// TIA Portal V17 export
// export: Created 2025-03-07T09:19:54.7926162Z, ExportSetting WithDefaults, DisplayName Totally Integrated Automation Portal, DisplayVersion V17 Update 8, DisplayName TIA Portal Openness, DisplayVersion V17 Update 8, DisplayName TIA Portal Version Control Interface, DisplayVersion V17, DisplayName SINAMICS Startdrive Advanced, DisplayVersion V17 SP2, DisplayName SINAMICS Startdrive G110M, G120, G120C, G120D, G120P, G115D, DisplayVersion V17 SP2, DisplayName SINAMICS Startdrive G130, G150, S120, S150, SINAMICS MV, S210, DisplayVersion V17 SP2, DisplayName STEP 7 Professional, DisplayVersion V17 Update 8, DisplayName SINUMERIK ONE STEP 7 Toolbox, DisplayVersion V17 Update 12, DisplayName SINUMERIK 840D sl STEP 7 Toolbox, DisplayVersion V17 Update 12, DisplayName STEP 7 Safety, DisplayVersion V17 Update 6, DisplayName WinCC Advanced, DisplayVersion V17 Update 8
TYPE "ABB_OUTPUTS"
// stored: IsFailsafeCompliant false
   STRUCT
      SYSTEM_SIGNAL : Struct
         SYS_MOTOR_ON : Bool;   // MACHINE HEARTBEAT (MACHINE TO GANTRY) / MOTORS ON STATE
         SYS_MOTOR_OFF : Bool;   // MOTORS OFF STATE
         SYS_CYCLE_ON : Bool;   // MACHINE EMERGENCY STOP OK (MACHINE TO GANTRY) / ROBOT IN CYCLE ON STATE
         SYS_AUTO_ON : Bool;   // MACHINE SAFETY GATES OK (LOCKED)(MACHINE TO GANTRY) / ROBOT IN AUTO MODE
         SYS_EMERG_UOP : Bool;   // MACHINE IN MANUAL MODE (MACHINE TO GANTRY) / EMERGENCY STOP ACTIVE
         SYS_ERROR : Bool;   // MACHINE IN AUTO MODE(MACHINE TO GANTRY) / EXECUTION ERROR ACTIVE
         SPARE_0_6 : Bool;   // MACHINE AUTO CYCLE RUNNING (MACHINE TO GANTRY)
         SPARE_0_7 : Bool;   // MACHINE IS IN WARMUP CYCLE (MACHINE TO GANTRY)
         SPARE_1_0 : Byte;   // MACHINE IN RUN OUT MODE (MACHINE TO GANTRY)
         SPARE_2_0 : Byte;   // MACHINE PART DEMAND SOON (MACHINE TO GANTRY)
         SPARE_3_0 : Byte;
      END_STRUCT;
      GENERAL_SIGNAL : Struct
         STYLE_INIT_ACK : Bool;   // GANTRY HEARTBEAT (GANTRY TO MACHINE) / ACKNOWLEDGE INITIATE STYLE
         IN_CYCLE : Bool;   // IN CYCLE
         REQ_TO_CONT : Bool;   // GANTRY EMERGENCY STOP OK (GANTRY TO MACHINE) / REQUEST TO CONTINUE
         DRY_CYCLE : Bool;   // DRY CYCLE MODE
         RBT_100_SPD : Bool;   // GANTRY IN MANUAL MODE (GANTRY TO MACHINE) / ROBOT 100% SPEED
         RBT_HEARTBEAT : Bool;   // GANTRY IN AUTO MODE (GANTRY TO MACHINE) / ROBOT HEARTBEAT SIGNAL
         "OP_PANEL_E-STOP" : Bool;   // GANTRY IN AUTO CYCLE RUNNING (GANTRY TO MACHINE) / OPERATOR PANEL E-STOP
         "TEACH_PENDANT_E-STOP" : Bool;   // GANTRY OVERHEAD DOOR CLOSED & LOCKED (GANTRY TO MACHINE) / TEACH PENDANT E-STOP
         EXT_ENABLED : Bool;   // GANTRY IN RUN OUT COMPLETE(GANTRY TO MACHINE) / EXTERNAL E-STOP
         DEAD_ENABLED : Bool;   // GANTRY CLEAR OF MACHINE (GANTRY TO MACHINE) / DEADMAN E-STOP
         "I/O_SIMULATE" : Bool;   // GANTRY CLEAR OF FIXTURE (GANTRY TO MACHINE) / I/O SIMULATED
         SRV_DISC_OFF : Bool;   // SERVO DISABLED OFF
         SRV_BATT_ALARM : Bool;   // LOW BATTERY ALARM ON SERVO
         TASK_OK : Bool;   // TASK OK
         STEP_MODE_ON : Bool;   // STEP MODE STATUS
         AUTO_MODE_ON : Bool;   // SELECTOR SWITCH IS SET TO AUTO
         MANUAL_ON : Bool;   // SELECTOR SWITCH IS SET TO MANUAL
         FENCE_OPEN : Bool;   // FENCE IS OPEN
         INTERLOCK : Bool;   // ROBOT IN INTERLOCK
         ROUT_ACTIVE : Bool;   // ROUTER ACTIVE BIT
         FAULT_RSP_ACK : Bool;   // HMI OPTION FAULT RESPONSE
         DCS_SIGN_MATCH : Bool;   // DCS SIGNATURE MATCH
         REQ_DEC_CODE : Bool;   // REQUEST DECITION
         FLT_TASK_UOPPED : Bool;   // ROBOT TASK STOPPED
         FLT_COLLISION : Bool;   // ROBOT COLLITION FAULT
         FLT_BAD_PLC_INPUT : Bool;   // BAD PLC INPUT
         FLT_GRIP_LOW_PRS : Bool;   // ROBOT GRIPPER PRESSURE LOW
         FLT_BAD_OPTN : Bool;   // BAD PLC FAULT RESPONSE
         RECOV_AT_MAIN : Bool;   // RECOVERY POINTER TO MAIN
         FLT_USER_BIT_8 : Bool;   // USER DEFINABLE FAULT BIT
         SPARE_7_6 : Bool;
         SPARE_7_7 : Bool;
         SPARE_8_0 : Byte;
         SPARE_9_0 : Byte;
      END_STRUCT;
      PROGRAM : Struct
         STYLE_PROGRAM_ACK : Byte;   // GANTRY HEARTBEAT (GANTRY TO MACHINE) / SELECT STYLE PROGRAM ACKNOWLEDGE
         DEC_CODE_ACK : Byte;   // SELECT DECITION CODE ACKNOWLEDGE
         PART_TYPE_ACK : Byte;   // GANTRY EMERGENCY STOP OK (GANTRY TO MACHINE) / PART TYPE ACKNOWLEDGE
         SPARE_13_0 : Byte;   // GANTRY EMERGENCY STOP OK (GANTRY TO MACHINE)
      END_STRUCT;
      GRIPPERS : Struct
         T1_GRIPPER_A_OPEN_REQ : Bool;   // ROBOT TOOL 1 GRIPPER A OPEN REQUEST
         T1_GRIPPER_A_CLOSE_REQ : Bool;   // ROBOT TOOL 1 GRIPPER A CLOSE REQUEST
         SPARE_14_2 : Bool;
         SPARE_14_3 : Bool;
         T1_GRIPPER_A_OPEN : Bool;   // ROBOT TOOL 1 GRIPPER A OPEN
         T1_GRIPPER_A_CLOSED : Bool;   // ROBOT TOOL 1 GRIPPER A CLOSED
         SPARE_14_6 : Bool;
         SPARE_14_7 : Bool;
         T1_GRIPPER_B_OPEN_REQ : Bool;   // ROBOT TOOL 1 GRIPPER B OPEN REQUEST
         T1_GRIPPER_B_CLOSE_REQ : Bool;   // ROBOT TOOL 1 GRIPPER B CLOSE REQUEST
         SPARE_15_2 : Bool;
         SPARE_15_3 : Bool;
         T1_GRIPPER_B_OPEN : Bool;   // ROBOT TOOL 1 GRIPPER B OPEN
         T1_GRIPPER_B_CLOSED : Bool;   // ROBOT TOOL 1 GRIPPER B CLOSED
         SPARE_15_6 : Bool;
         SPARE_15_7 : Bool;
         T1_GRIPPER_C_OPEN_REQ : Bool;   // ROBOT TOOL 1 GRIPPER C OPEN REQUEST
         T1_GRIPPER_C_CLOSE_REQ : Bool;   // ROBOT TOOL 1 GRIPPER C CLOSE REQUEST
         SPARE_16_2 : Bool;
         SPARE_16_3 : Bool;
         T1_GRIPPER_C_OPEN : Bool;   // ROBOT TOOL 1 GRIPPER C OPEN
         T1_GRIPPER_C_CLOSED : Bool;   // ROBOT TOOL 1 GRIPPER C CLOSED
         SPARE_16_6 : Bool;
         SPARE_16_7 : Bool;
         T1_GRIPPER_D_OPEN_REQ : Bool;   // ROBOT TOOL 1 GRIPPER D OPEN REQUEST
         T1_GRIPPER_D_CLOSE_REQ : Bool;   // ROBOT TOOL 1 GRIPPER D CLOSE REQUEST
         SPARE_17_2 : Bool;
         SPARE_17_3 : Bool;
         T1_GRIPPER_D_OPEN : Bool;   // ROBOT TOOL 1 GRIPPER D OPEN
         T1_GRIPPER_D_CLOSED : Bool;   // ROBOT TOOL 1 GRIPPER D CLOSED
         SPARE_17_6 : Bool;
         SPARE_17_7 : Bool;
         T1_GRIPPER_E_OPEN_REQ : Bool;   // ROBOT TOOL 1 GRIPPER E OPEN REQUEST
         T1_GRIPPER_E_CLOSE_REQ : Bool;   // ROBOT TOOL 1 GRIPPER E CLOSE REQUEST
         SPARE_18_2 : Bool;
         SPARE_18_3 : Bool;
         T1_GRIPPER_E_OPEN : Bool;   // ROBOT TOOL 1 GRIPPER E OPEN
         T1_GRIPPER_E_CLOSED : Bool;   // ROBOT TOOL 1 GRIPPER E CLOSED
         SPARE_18_6 : Bool;
         SPARE_18_7 : Bool;
         T2_GRIPPER_A_OPEN_REQ : Bool;   // ROBOT TOOL 2 GRIPPER A OPEN REQUEST
         T2_GRIPPER_A_CLOSE_REQ : Bool;   // ROBOT TOOL 2 GRIPPER A CLOSE REQUEST
         SPARE_19_2 : Bool;
         SPARE_19_3 : Bool;
         T2_GRIPPER_A_OPEN : Bool;   // ROBOT TOOL 2 GRIPPER A OPEN
         T2_GRIPPER_A_CLOSED : Bool;   // ROBOT TOOL 2 GRIPPER A CLOSED
         SPARE_19_6 : Bool;
         SPARE_19_7 : Bool;
         T2_GRIPPER_B_OPEN_REQ : Bool;   // ROBOT TOOL 2 GRIPPER B OPEN REQUEST
         T2_GRIPPER_B_CLOSE_REQ : Bool;   // ROBOT TOOL 2 GRIPPER B CLOSE REQUEST
         SPARE_20_2 : Bool;
         SPARE_20_3 : Bool;
         T2_GRIPPER_B_OPEN : Bool;   // ROBOT TOOL 2 GRIPPER B OPEN
         T2_GRIPPER_B_CLOSED : Bool;   // ROBOT TOOL 2 GRIPPER B CLOSED
         SPARE_20_6 : Bool;
         SPARE_20_7 : Bool;
         T2_GRIPPER_C_OPEN_REQ : Bool;   // ROBOT TOOL 2 GRIPPER C OPEN REQUEST
         T2_GRIPPER_C_CLOSE_REQ : Bool;   // ROBOT TOOL 2 GRIPPER C CLOSE REQUEST
         SPARE_21_2 : Bool;
         SPARE_21_3 : Bool;
         T2_GRIPPER_C_OPEN : Bool;   // ROBOT TOOL 2 GRIPPER C OPEN
         T2_GRIPPER_C_CLOSED : Bool;   // ROBOT TOOL 2 GRIPPER C CLOSED
         SPARE_21_6 : Bool;
         SPARE_21_7 : Bool;
         T2_GRIPPER_D_OPEN_REQ : Bool;   // ROBOT TOOL 2 GRIPPER D OPEN REQUEST
         T2_GRIPPER_D_CLOSE_REQ : Bool;   // ROBOT TOOL 2 GRIPPER D CLOSE REQUEST
         SPARE_22_2 : Bool;
         SPARE_22_3 : Bool;
         T2_GRIPPER_D_OPEN : Bool;   // ROBOT TOOL 2 GRIPPER D OPEN
         T2_GRIPPER_D_CLOSED : Bool;   // ROBOT TOOL 2 GRIPPER D CLOSED
         SPARE_22_6 : Bool;
         SPARE_22_7 : Bool;
         T2_GRIPPER_E_OPEN_REQ : Bool;   // ROBOT TOOL 2 GRIPPER E OPEN REQUEST
         T2_GRIPPER_E_CLOSE_REQ : Bool;   // ROBOT TOOL 2 GRIPPER E CLOSE REQUEST
         SPARE_23_2 : Bool;
         SPARE_23_3 : Bool;
         T2_GRIPPER_E_OPEN : Bool;   // ROBOT TOOL 2 GRIPPER E OPEN
         T2_GRIPPER_E_CLOSED : Bool;   // ROBOT TOOL 2 GRIPPER E CLOSED
         SPARE_23_6 : Bool;
         SPARE_23_7 : Bool;
         T1_ALL_GRIPS_OPEN_REQ : Bool;   // ROBOT TOOL 1 OPEN ALL GRIPPERS REQUEST
         T1_ALL_GRIPS_CLOSE_REQ : Bool;   // ROBOT TOOL 1 CLOSE ALL GRIPPERS REQUEST
         T1_ALL_GRIPPERS_OPEN : Bool;   // ROBOT TOOL 1 ALL GRIPPERS OPEN
         T1_ALL_GRIPPERS_CLOSED : Bool;   // ROBOT TOOL 1 ALL GRIPPERS CLOSED
         SPARE_24_4 : Bool;
         SPARE_24_5 : Bool;
         SPARE_24_6 : Bool;
         SPARE_24_7 : Bool;
         T2_ALL_GRIPS_OPEN_REQ : Bool;   // ROBOT TOOL 2 CLOSE ALL GRIPPERS REQUEST
         T2_ALL_GRIPS_CLOSE_REQ : Bool;   // ROBOT TOOL 2 CLOSE ALL GRIPPERS REQUEST
         T2_ALL_GRIPPERS_OPEN : Bool;   // ROBOT TOOL 2 ALL GRIPPERS OPEN
         T2_ALL_GRIPPERS_CLOSED : Bool;   // ROBOT TOOL 2 ALL GRIPPERS CLOSED
         SPARE_25_4 : Bool;
         SPARE_25_5 : Bool;
         SPARE_25_6 : Bool;
         SPARE_25_7 : Bool;
         SPARE_26_0 : Byte;
         FAULT_NUMBER : Byte;   // FAULT RESPONSE
      END_STRUCT;
      CLEARS : Struct
         CLEAR_U_1_ACK : Bool;   // GANTRY HEARTBEAT (GANTRY TO MACHINE) / CLEAR UNIT 1
         CLEAR_U_2_ACK : Bool;   // CLEAR UNIT 2
         CLEAR_U_3_ACK : Bool;   // GANTRY EMERGENCY STOP OK (GANTRY TO MACHINE) / CLEAR UNIT 3
         CLEAR_U_4_ACK : Bool;   // CLEAR UNIT 4
         CLEAR_U_5_ACK : Bool;   // GANTRY IN MANUAL MODE (GANTRY TO MACHINE) / CLEAR UNIT 5
         CLEAR_U_6_ACK : Bool;   // GANTRY IN AUTO MODE (GANTRY TO MACHINE) / CLEAR UNIT 6
         CLEAR_U_7_ACK : Bool;   // GANTRY IN AUTO CYCLE RUNNING (GANTRY TO MACHINE) / CLEAR UNIT 7
         CLEAR_U_8_ACK : Bool;   // GANTRY OVERHEAD DOOR CLOSED & LOCKED (GANTRY TO MACHINE) / CLEAR UNIT 8
         CLEAR_U_9_ACK : Bool;   // GANTRY IN RUN OUT COMPLETE(GANTRY TO MACHINE) / CLEAR UNIT 9
         CLEAR_U_10_ACK : Bool;   // GANTRY CLEAR OF MACHINE (GANTRY TO MACHINE) / CLEAR UNIT 10
         SPARE_29_2 : Bool;   // GANTRY CLEAR OF FIXTURE (GANTRY TO MACHINE)
         SPARE_29_3 : Bool;
         SPARE_29_4 : Bool;
         SPARE_29_5 : Bool;   // GANTRY PART TYPE CHANGE REQUESTED (GANTRY TO MACHINE)
         SPARE_29_6 : Bool;   // GANTRY REQUEST MACHINE TO RUN WITH LOADED PARTS (GANTRY TO MACHINE)
         SPARE_29_7 : Bool;   // GANTRY RUN OUT REQUESTED (GANTRY TO MACHINE)
         SPARE_30_0 : Byte;
         SPARE_31_0 : Byte;
      END_STRUCT;
      TASKS : Struct
         TSK_COMPLETED_1 : Bool;   // GANTRY HEARTBEAT (GANTRY TO MACHINE) / ROBOT TASK 1 COMPLETED
         TSK_COMPLETED_2 : Bool;   // ROBOT TASK 2 COMPLETED
         TSK_COMPLETED_3 : Bool;   // GANTRY EMERGENCY STOP OK (GANTRY TO MACHINE) / ROBOT TASK 3 COMPLETED
         TSK_COMPLETED_4 : Bool;   // ROBOT TASK 4 COMPLETED
         TSK_COMPLETED_5 : Bool;   // GANTRY IN MANUAL MODE (GANTRY TO MACHINE) / ROBOT TASK 5 COMPLETED
         TSK_COMPLETED_6 : Bool;   // GANTRY IN AUTO MODE (GANTRY TO MACHINE) / ROBOT TASK 6 COMPLETED
         TSK_COMPLETED_7 : Bool;   // GANTRY IN AUTO CYCLE RUNNING (GANTRY TO MACHINE) / ROBOT TASK 7 COMPLETED
         TSK_COMPLETED_8 : Bool;   // GANTRY OVERHEAD DOOR CLOSED & LOCKED (GANTRY TO MACHINE) / ROBOT TASK 8 COMPLETED
         SPARE_33_0 : Byte;   // GANTRY IN RUN OUT COMPLETE(GANTRY TO MACHINE) / ROBOT TASK 9 COMPLETED
         SPARE_34_0 : Byte;   // GANTRY CLEAR OF MACHINE (GANTRY TO MACHINE) / ROBOT TASK 10 COMPLETED
         SPARE_35_0 : Byte;   // GANTRY CLEAR OF FIXTURE (GANTRY TO MACHINE)
         SPARE_36_0 : Byte;
         SPARE_37_0 : Byte;
         SPARE_38_0 : Byte;
         SPARE_39_0 : Byte;
      END_STRUCT;
      POSITIONS : Struct
         HOME : Bool;   // GANTRY HEARTBEAT (GANTRY TO MACHINE) / ROBOT AT HOME POSITION
         MAINT : Bool;   // ROBOT AT MAINTENANCE POSITION
         REPAIR : Bool;   // GANTRY EMERGENCY STOP OK (GANTRY TO MACHINE) / ROBOT AT REPAIRED POSITION
         ALIGN : Bool;   // ROBOT AT ALIGNED POSITION
         SHIP : Bool;   // GANTRY IN MANUAL MODE (GANTRY TO MACHINE) / ROBOT AT SHIPPED POSITION
         SPARE_38_5 : Bool;   // GANTRY IN AUTO MODE (GANTRY TO MACHINE)
         SPARE_38_6 : Bool;   // GANTRY IN AUTO CYCLE RUNNING (GANTRY TO MACHINE)
         SPARE_38_7 : Bool;   // GANTRY OVERHEAD DOOR CLOSED & LOCKED (GANTRY TO MACHINE)
         UNIT_1 : Bool;   // GANTRY OVERHEAD DOOR CLOSED & LOCKED (GANTRY TO MACHINE) / ROBOT AT POUNCE POSITION UNIT 1
         UNIT_2 : Bool;   // GANTRY OVERHEAD DOOR CLOSED & LOCKED (GANTRY TO MACHINE) / ROBOT AT POUNCE POSITION UNIT 2
         UNIT_3 : Bool;   // GANTRY OVERHEAD DOOR CLOSED & LOCKED (GANTRY TO MACHINE) / ROBOT AT POUNCE POSITION UNIT 3
         UNIT_4 : Bool;   // GANTRY OVERHEAD DOOR CLOSED & LOCKED (GANTRY TO MACHINE) / ROBOT AT POUNCE POSITION UNIT 4
         UNIT_5 : Bool;   // GANTRY OVERHEAD DOOR CLOSED & LOCKED (GANTRY TO MACHINE) / ROBOT AT POUNCE POSITION UNIT 5
         UNIT_6 : Bool;   // GANTRY IN RUN OUT COMPLETE(GANTRY TO MACHINE) / ROBOT AT POUNCE POSITION UNIT 6
         UNIT_7 : Bool;   // GANTRY IN RUN OUT COMPLETE(GANTRY TO MACHINE) / ROBOT AT POUNCE POSITION UNIT 7
         UNIT_8 : Bool;   // GANTRY IN RUN OUT COMPLETE(GANTRY TO MACHINE) / ROBOT AT POUNCE POSITION UNIT 8
         SPARE_42_0 : Byte;   // GANTRY CLEAR OF MACHINE (GANTRY TO MACHINE)
         SPARE_43_0 : Byte;   // GANTRY CLEAR OF FIXTURE (GANTRY TO MACHINE)
         SPARE_44_0 : Byte;
         SPARE_45_0 : Byte;
      END_STRUCT;
      SPARES : Array[46..63] of Byte;
   END_STRUCT;
END_TYPE
